FUNCTION_BLOCK Temperature_Ctr
VAR_INPUT
	actual_tem : REAL;
	limit_tem : REAL;
	th : REAL;
	Enable : BOOL;	
	
	//relief_turn : BOOL := FALSE;	
   
	
END_VAR
VAR_OUTPUT
	Power_Fan :BOOL;
END_VAR
VAR
	A : REAL;
	B : REAL;
	
END_VAR


IF Enable = TRUE THEN 
	A := limit_tem-th;
	B := limit_tem +th;
	
	IF (actual_tem <= A)  THEN 
		Power_Fan := FALSE;
	ELSIF (actual_tem >= B) THEN
		Power_Fan := TRUE;
	END_IF
END_IF

END_FUNCTION_BLOCK

(* stored: Version 1.1.0.1, ProductVersion 3.1.4024.4
   POU Temperature_Ctr: Id {cee14709-947c-49ab-a6d8-a97143dd7e34}, SpecialFunc None *)
